{attribute 'GeneratedUsingTerminal: KL8610-0001'}
{attribute addProperty BoxType "KL8610-0001"}
{attribute addProperty Id "KL8601_1AT %Q*KL_6576A6810KL8601_2AT %Q*KL_6576A6810"}
{attribute addProperty CRC "1518594124"}
{attribute addProperty Size "0"}
TYPE KL_5A83E84C :
STRUCT
	{attribute addProperty Name "KL8601_1"}
	KL8601_1 : KL_6576A681;
	{attribute addProperty Name "KL8601_2"}
	KL8601_2 : KL_6576A681;
END_STRUCT
END_TYPE

(* stored: Version 1.2.0.0, ProductVersion 3.1.4024.9
   DUT KL_5A83E84C: Id {65d89a5f-8802-48a3-beb0-2bac37b516f5} *)
